TYPE E_ModeMMA :
(
	Init := 0,
	Auto,
	Man
);
END_TYPE

(* stored: Version 1.1.0.1, ProductVersion 3.1.4020.6
   DUT E_ModeMMA: Id {f5b067f7-751c-4839-a931-c6db6ef3a31f} *)
